FUNCTION_BLOCK FB_Profiler
VAR_INPUT
END_VAR
VAR_OUTPUT
END_VAR
VAR
	fbProfiler:		Profiler;
END_VAR

METHOD PUBLIC M_Reset : BOOL
VAR_INPUT
END_VAR
fbProfiler(START:= false, RESET:= True);
END_METHOD

METHOD PUBLIC M_Restart : BOOL
VAR_INPUT
END_VAR
fbProfiler(START:= True, RESET:= FALSE);
END_METHOD

METHOD PUBLIC M_Start : BOOL
VAR_INPUT
END_VAR
fbProfiler(START:= True, RESET:= FALSE);
END_METHOD

PROPERTY PUBLIC P_Busy : bool
GET
P_Busy:= fbProfiler.BUSY;
END_GET
END_PROPERTY

END_FUNCTION_BLOCK

(* stored: Version 1.1.0.1
   POU FB_Profiler: Id {c14cfb6c-09fa-013d-01ad-5952a1bb49b2}, SpecialFunc None
   Method M_Reset: Id {1cb04307-072a-068a-08e9-e6c0b54e48e8}
   Method M_Restart: Id {06d22935-012a-0ff6-08f3-d2ffe893a5c3}
   Method M_Start: Id {b0d529f8-0646-0c38-2bb5-7235169dde15}
   Property P_Busy: Id {146312e2-1031-06cd-3fe8-ea7f1db13c6f}
   Get Get: Id {620d4dce-97f9-051f-17f8-5298f3b6fbcb} *)
